(* IEC 61131-3 sources: volt/packages/volt-lsp-iec/test-corpus/lenze-mid/Device/Plc Logic/Application/A70_MachineModuleSources/MM_MachineControl/ATF_ADS, 5 files *)

(* ---- fc_CheckNumberOfErrorsRegister.pou ---- *)
FUNCTION fc_CheckNumberOfErrorsRegister : bool
VAR_INPUT
	iPositie			: ARRAY[0..CTE.ct_ArraySizeCheckRegister] OF cUDT_ShiftRegister_Positie;
	iPositionToCheck : INT;
	iAmountOfErrors : INT;

END_VAR
VAR
	tAmountError : INT;
	tLastPositionToCheck : INT;
	tIndex : INT;

END_VAR
VAR_IN_OUT
	//ioPositie			: ARRAY[0..CTE.ct_ArraySizeCheckRegister] OF cUDT_ShiftRegister_Positie;

END_VAR
VAR_OUTPUT
	oError	: BOOL;
END_VAR
%LANGUAGE ST
//Init
oError := FALSE;
tLastPositionToCheck := 0;
tAmountError := 0;

tLastPositionToCheck := iPositionToCheck + iAmountOfErrors;

FOR tIndex := iPositionToCheck TO tLastPositionToCheck DO

    IF iPositie[tIndex].Infeed.Cigar_Present_Infeed  THEN
        IF iPositie[tIndex].Outfeed.Cigar_Present_Outfeed = 0 THEN
            tAmountError := tAmountError + 1;
        END_IF;
    END_IF;

    IF tAmountError >= iAmountOfErrors THEN
        oError := TRUE;
        EXIT; //Exit for loop
    END_IF;

END_FOR;

END_FUNCTION

(* ---- fc_MeanValue.pou ---- *)
FUNCTION fc_MeanValue
VAR_INPUT
	iLength						: INT;
	iAcquireNewValue			: BOOL;
	iNewValue					: INT;

END_VAR

VAR_OUTPUT
	oMeanValue					: INT;
END_VAR

VAR
	tIndex						: INT;
	tMean						: DINT;
	tCountToIndexNumber			: INT;

END_VAR

VAR_IN_OUT
	ioValues					: ARRAY[0..50] OF INT;
END_VAR
%LANGUAGE ST
oMeanValue := 0;
tMean := 0;
tCountToIndexNumber := iLength - 2; //count from 0 to length -1, but shift is 1 index less -> -2

FOR tIndex:=tCountToIndexNumber TO 0 BY -1 DO
    ioValues[tIndex + 1] := ioValues[tIndex];
    tMean := tMean + ioValues[tIndex];

    IF tIndex= 0 THEN
        ioValues[0] := iNewValue;
        tMean := tMean + ioValues[tIndex];
    END_IF;

END_FOR;
oMeanValue := DINT_TO_INT(tMean / iLength);

END_FUNCTION

(* ---- fc_ShiftRegister.pou ---- *)
FUNCTION fc_ShiftRegister : bool
VAR_INPUT
END_VAR
VAR
	i: INT;
END_VAR
VAR_IN_OUT
	//ioPositie			: ARRAY[0..CTE.ct_ArraySizeCheckRegister] OF cUDT_ShiftRegister_Positie;
	ioPositie			: ARRAY[0..CTE.ct_ArraySizeCheckRegister] OF cUDT_ShiftRegister_Positie;
END_VAR
%LANGUAGE ST
(*
    Shift register
*)
FOR i := CTE.ct_ArraySizeCheckRegister TO 2 BY -1 DO
    ioPositie[i] := ioPositie[i - 1];
END_FOR;

//Eerste register leegmaken
ioPositie[1] := db_CheckRegister.EmptyCheckRegister;

END_FUNCTION

(* ---- Dryer.pou ---- *)
FUNCTION_BLOCK Dryer
VAR_INPUT
	iGenFlags : UDT_GeneralFlags;
iMachineStarted : Bool;
iSwitchDryer : Bool;
iDryerClosed : Bool;
iStartFeedForward : Bool;
iStopFeedForward : Bool;
iPermissionDownstream : Bool;
iSetPowerHeater1 : Int;
iSetPowerHeater2 : Int;
iSetPowerHeater3 : Int;
iPowerOrAnalog : Bool;
iSpeedForEmptying : INT;

END_VAR
VAR_OUTPUT
	ENO: BOOL;
	oFeedForward : BOOL;
oEnableHeaters : Bool;
oPowerHeater1 : Word;
oPowerHeater2 : Word;
oPowerHeater3 : Word;
oFaultDryerOpened : Bool;

END_VAR
VAR
	tEmptyingCycleInterval : DINT;

	stAuxFeedForward: rs;
	tConditionHeaterTimeOut: BOOL;
	tEnableHeaters: BOOL;
	stActPowerHeater1: INT;
	stActPowerHeater2: INT;
	stActPowerHeater3: INT;
	TMR_DryerOpened: TON;
END_VAR

VAR RETAIN PERSISTENT
	stReFeedForward: R_TRIG;
	TMR_IntervalTimerEmptying: TON;
	stFaultDryerOpened: sr;
	stReStopFeedForward: R_TRIG;
	TMR_HeaterTimeOut: TON;
END_VAR
%LANGUAGE LD
%NETWORK "DONE Network 1: Convert speed to cycle time"
// tEmtyingCycle : (1/(MachineSpeed/60))*1000 gives time in [ms]
EXECUTE(EN := RAIL(), 'tEmptyingCycleInterval:=(60*1000)/TO_DINT(iSpeedForEmptying);
');
%NETWORK "DONE Network 2: Feed forward dryer"
ASSIGN(stAuxFeedForward(SET := iStartFeedForward OR TMR_IntervalTimerEmptying(IN := ASSIGN(NOT(stReFeedForward(CLK := stAuxFeedForward.Q1)), Q => tConditionHeaterTimeOut), PT := OPERAND('DINT_TO_TIME(tEmptyingCycleInterval)')) AND iMachineStarted AND INVERT(stFaultDryerOpened.Q1) AND Mach1.GenFlags.DelayAfterSTO AND INVERT(iGenFlags.DriveIsRunning) AND iPermissionDownstream, RESET1 := stReStopFeedForward(CLK := iStopFeedForward)), Q => oFeedForward);
%NETWORK "DONE Network 3: Enable heaters"
VAR w1 : ANY; w2 : ANY; END_VAR
w1 := TRUE;
TMR_HeaterTimeOut(IN := w1 AND INVERT(LST_InputsOutputs.I133_1_PROX_zero_position_transport_ADS), PT := T#7S);
w2 := w1 AND iGenFlags.EnableAuxDrive AND iPermissionDownstream AND INVERT(TMR_HeaterTimeOut.Q) AND iSwitchDryer;
ASSIGN(w2, Q => oEnableHeaters);
ASSIGN(w2, Q => tEnableHeaters);
%NETWORK "DONE Network 4: Output power heater 1"
VAR w3 : ANY; w4 : ANY; END_VAR
w3 := True;
MOVE(EN := w3 AND INVERT(tEnableHeaters), 0, OUT => stActPowerHeater1);
w4 := w3 AND tEnableHeaters;
ADD(EN := w4 AND LST_General.Imp100ms, stActPowerHeater1, 10, OUT => stActPowerHeater1);
MOVE(EN := GT(EN := w4, stActPowerHeater1, iSetPowerHeater1).OUT, iSetPowerHeater1, OUT => stActPowerHeater1);
EXECUTE(EN := w3 AND INVERT(iPowerOrAnalog), 'oPowerHeater1:=INT_TO_WORD(stActPowerHeater1*27648/1000);

');
MOVE(EN := w3 AND iPowerOrAnalog, OPERAND('INT_TO_WORD(stActPowerHeater1)'), OUT => oPowerHeater1);
%NETWORK "DONE Network 5: Output power heater 2"
VAR w5 : ANY; w6 : ANY; END_VAR
w5 := True;
MOVE(EN := w5 AND INVERT(tEnableHeaters), 0, OUT => stActPowerHeater2);
w6 := w5 AND tEnableHeaters;
ADD(EN := w6 AND LST_General.Imp100ms, stActPowerHeater2, 10, OUT => stActPowerHeater2);
MOVE(EN := GT(EN := w6, stActPowerHeater2, iSetPowerHeater2).OUT, iSetPowerHeater2, OUT => stActPowerHeater2);
EXECUTE(EN := w5 AND INVERT(iPowerOrAnalog), 'oPowerHeater2:=INT_TO_WORD(stActPowerHeater2*27648/1000);

');
MOVE(EN := w5 AND iPowerOrAnalog, OPERAND('INT_TO_WORD(stActPowerHeater2)'), OUT => oPowerHeater2);
%NETWORK "DONE Network 6: Output power heater 3"
VAR w7 : ANY; w8 : ANY; END_VAR
w7 := True;
MOVE(EN := w7 AND INVERT(tEnableHeaters), 0, OUT => stActPowerHeater3);
w8 := w7 AND tEnableHeaters;
ADD(EN := w8 AND LST_General.Imp100ms, stActPowerHeater3, 10, OUT => stActPowerHeater3);
MOVE(EN := GT(EN := w8, stActPowerHeater3, iSetPowerHeater3).OUT, iSetPowerHeater3, OUT => stActPowerHeater3);
EXECUTE(EN := w7 AND INVERT(iPowerOrAnalog), 'oPowerHeater3:=INT_TO_WORD(stActPowerHeater3*27648/1000);

');
MOVE(EN := w7 AND iPowerOrAnalog, OPERAND('INT_TO_WORD(stActPowerHeater3)'), OUT => oPowerHeater3);
%NETWORK "DONE Network 37: Fault: dryer opened"
ASSIGN(stFaultDryerOpened(SET1 := TMR_DryerOpened(IN := iMachineStarted AND iSwitchDryer AND INVERT(iDryerClosed) AND INVERT(stFaultDryerOpened.Q1), PT := T#5S), RESET := iGenFlags.StartFlag), Q => oFaultDryerOpened);
%NETWORK
ASSIGN(RAIL(), Q => ENO);

END_FUNCTION_BLOCK

(* ---- TrayFiller.pou ---- *)
FUNCTION_BLOCK TrayFiller
VAR_INPUT
	iGenFlags : UDT_GeneralFlags;
iMachineStarted : Bool;
iButtonChangeTray : Bool;
iButtonTrayDown : Bool;
iButtonTrayUp : Bool;
iCigarAtCrossover : Bool;
iStartFeedForward : Bool;
iStopFeedForward : Bool;
iCigarAtInpusher : Bool;
iRpsInpusher : Bool;
iEpsInpusher : Bool;
iGuardInpusher : Bool;
iPsElevatorUp : Bool;
iPsElevatorDown : Bool;
iPulseCounterElevator : Bool;
iFcGuardTrayOnElev : Bool;
iRowHeight : Int;
iSetNumberOfRows : Int;
iInitialDescentValue : Int;
iLightCurtainInpusher : Bool;
iLightCurtainElevator : Bool;
iPsInfeedConvAtInit : Bool;
iPsInfeedConvAtElev : Bool;
iFcGuardTrayFromElev : Bool;
iFcOutfeedConvFull : Bool;
iTestProd : Bool;

END_VAR
VAR_OUTPUT
	oValveInpusher : BOOL;
oValveTiltInpusher : Bool;
oFeedForwardMotor : Bool;
oElevatorMotorUp : Bool;
oElevatorMotorDown : Bool;
oElevatorMotorBrake : Bool;
oOutfeedMotorFwd : Bool;
oInfeedMotorFwd : Bool;
oInfeedMotorRev : Bool;

END_VAR
VAR
	stRestposition : BOOL;
stInpushingRow : Bool;
stDecendTray : Bool;
stTrayDecended : Bool;
stTiltInpusher : Bool;
stReturnInpusher : Bool;
stLowerInpusher : Bool;
stMoveElevatorUp : Bool;
stMoveElevatorDown : Bool;
stSrCigarAtEndBeforeLast : Bool;
stSrCigarAtEnd : Bool;
stReStopFeedForward : r_trig;
stAuxFeedForward : RS;
stRePulseCounter : r_trig;
stFePulseCounter : F_TRIG;
stFaultInpusherBlocked : SR;
stFaultPositionTray : SR;
stActHeightElevator : Int;
stLightCurtainInterruptedBeforeStart : Bool;
stLightCurtainInterruptedDuringInpushing : Bool;
stElevatorAtBottom : Bool;
stOutfeedTray : Bool;
stOutfeedConvFull : Bool;
stTrayFaultOutfeeding : Bool;
stTrayFedOut : Bool;
stElevatorAtTop : Bool;
stInfeedTray : Bool;
bReturnInfeedConv : Bool;
bFaultOutfeeding : Bool;
bRecoverFromLightCurtainInterrupted : Bool;
TMR_InpusherDown : ton;
TMR_DelayReturnInfeed : ton;
TMR_DelayDescend : ton;
TMR_InpusherTilted : ton;
TMR_DelayEmptying : ton;
TMR_DelayFaultOutfeed : ton;
TMR_DelayTrayFedOut : ton;
TOdoTEst : ctd;

	tBool: BOOL;
	tInt: INT;
	SET_stFaultPositionTray:BOOL;
END_VAR

VAR_IN_OUT
	ioActNumberOfRows: INT;
END_VAR
%LANGUAGE LD
%NETWORK "DONE NETWORK 1: Condition: Reset all"
ASSIGN(LST_General.FirstCycle, Q_SET => stRestposition, Q_RESET => bReturnInfeedConv, Q_RESET => stInpushingRow, Q_RESET => stDecendTray, Q_RESET => stTrayDecended, Q_RESET => stTiltInpusher, Q_RESET => stReturnInpusher, Q_RESET => stLowerInpusher, Q_RESET => stMoveElevatorUp, Q_RESET => stMoveElevatorDown, Q_RESET => stElevatorAtBottom, Q_RESET => stOutfeedTray, Q_RESET => stTrayFedOut, Q_RESET => stElevatorAtTop, Q_RESET => stInfeedTray, Q_RESET => stLightCurtainInterruptedBeforeStart, Q_RESET => stLightCurtainInterruptedDuringInpushing, Q_RESET => stTrayFaultOutfeeding, Q_RESET => bRecoverFromLightCurtainInterrupted, Q_RESET => stSrCigarAtEnd);
%NETWORK "DONE NETWORK 2: Condition: Rest position"
VAR w1 : ANY; END_VAR
w1 := TMR_InpusherDown(IN := stLowerInpusher, PT := T#500MS) OR stInfeedTray AND iPsInfeedConvAtElev OR stLightCurtainInterruptedBeforeStart AND iLightCurtainInpusher AND iGenFlags.StartFlag;
ASSIGN(w1, Q_SET => stRestposition, Q_RESET => stLowerInpusher, Q_RESET => stInfeedTray, Q_RESET => stLightCurtainInterruptedBeforeStart);
ASSIGN(w1 AND INVERT(iFcGuardTrayOnElev) AND iTestProd, Q_SET => Trayfiller_Data.Alarms.AlmTrayInfeeding);
%NETWORK "TODO NETWORK 3: Condition: Set infeed conveyor at init position"
VAR w2 : ANY; END_VAR
w2 := True;
ASSIGN(w2 AND bReturnInfeedConv AND iPsInfeedConvAtInit, Q_RESET => bReturnInfeedConv);
ASSIGN(w2 AND iGenFlags.StartFlag AND (iFcGuardTrayOnElev OR INVERT(iTestProd)), Q_RESET => Trayfiller_Data.Alarms.AlmTrayInfeeding);
%NETWORK "DONE NETWORK 4: Delay return infeed conveyor"
TMR_DelayReturnInfeed(IN := bReturnInfeedConv, PT := T#500MS);
%NETWORK "DONE NETWORK 5: Condition: Inpushing row"
ASSIGN(stRestposition AND stSrCigarAtEnd AND INVERT(stFaultPositionTray.Q1), Q_SET => stInpushingRow, Q_RESET => stRestposition);
%NETWORK "TODO NETWORK 6: Condition: Light curtain inpusher interrupted before start"
ASSIGN((stInpushingRow OR stRestposition AND stSrCigarAtEndBeforeLast) AND INVERT(iLightCurtainInpusher) AND iRpsInpusher, Q_SET => stLightCurtainInterruptedBeforeStart, Q_RESET => stInpushingRow);
%NETWORK "TODO NETWORK 7: Condition: Decend tray"
ASSIGN(ADD(EN := (TMR_DelayDescend(IN := stInpushingRow AND iLightCurtainInpusher AND iEpsInpusher, PT := T#500MS) OR stLightCurtainInterruptedDuringInpushing AND iLightCurtainInpusher AND iGenFlags.StartFlag) AND INVERT(stFaultInpusherBlocked.Q1), ioActNumberOfRows, 1, OUT => ioActNumberOfRows), Q_SET => stDecendTray, Q_RESET => stInpushingRow, Q_RESET => stLightCurtainInterruptedDuringInpushing, Q_RESET => stSrCigarAtEndBeforeLast, Q_RESET => stSrCigarAtEnd);
%NETWORK "TODO NETWORK 8: Condition: Light curtain inpusher interrupted during inpushing"
ASSIGN(stInpushingRow AND INVERT(iLightCurtainInpusher) AND INVERT(iRpsInpusher), Q_SET => stLightCurtainInterruptedDuringInpushing, Q_RESET => stInpushingRow, Q_RESET => bRecoverFromLightCurtainInterrupted);
%NETWORK "TODO NETWORK 9: Condition: Tray decend"
VAR w3 : ANY; w4 : ANY; w5 : ANY; END_VAR
w3 := True;
w4 := w3 AND True;
w5 := w4 AND iPulseCounterElevator;
ASSIGN(stRePulseCounter(CLK := w5), Q => tBool);
ASSIGN(stFePulseCounter(CLK := w5), Q_SET => tBool);
ADD(EN := w4 AND tBool AND (stDecendTray OR stTrayDecended OR stTiltInpusher), stActHeightElevator, 5, OUT => stActHeightElevator);
ASSIGN(BRANCH_SHORTCIRCUIT(FEED := ADD(EN := MUL(EN := w3 AND stDecendTray, ioActNumberOfRows, iRowHeight, OUT => tInt), tInt, iInitialDescentValue, OUT => tInt), GE(EN := RAIL(), stActHeightElevator, tInt).OUT, iPsElevatorDown), Q_SET => stTrayDecended, Q_RESET => stDecendTray);
%NETWORK "TODO NETWORK 10: Condition: Tilt inpusher"
ASSIGN(stTrayDecended, Q_SET => stTiltInpusher, Q_RESET => stTrayDecended, Q_SET => bReturnInfeedConv);
%NETWORK "TODO NETWORK 11: Condition: Return inpusher"
ASSIGN(TMR_InpusherTilted(IN := stTiltInpusher, PT := T#500MS), Q_SET => stReturnInpusher, Q_RESET => stTiltInpusher);
%NETWORK "TODO NETWORK 12: Condition: Lower inpusher"
ASSIGN(LT(EN := stReturnInpusher AND iRpsInpusher, ioActNumberOfRows, iSetNumberOfRows).OUT AND INVERT(iPsElevatorDown) AND INVERT(stFaultInpusherBlocked.Q1), Q_SET => stLowerInpusher, Q_RESET => stReturnInpusher, Q_RESET => bRecoverFromLightCurtainInterrupted);
%NETWORK "TODO NETWORK 13: Condition: Move elevator down"
ASSIGN(BRANCH_SHORTCIRCUIT(BRANCH_SHORTCIRCUIT(FEED := stReturnInpusher AND iRpsInpusher, GE(EN := RAIL(), ioActNumberOfRows, iSetNumberOfRows).OUT, iPsElevatorDown) AND INVERT(stFaultInpusherBlocked.Q1) AND iMachineStarted, stOutfeedConvFull AND iGenFlags.StartFlag, TMR_DelayEmptying(IN := stRestposition AND iGenFlags.DelayAfterEmergStop AND iPsElevatorDown, PT := T#2S)), Q_SET => stMoveElevatorDown, Q_RESET => stReturnInpusher, Q_RESET => stOutfeedConvFull, Q_RESET => stRestposition);
%NETWORK "TODO NETWORK 14: Condition: Elevator at bottom"
ASSIGN(stMoveElevatorDown AND iPsElevatorDown OR stTrayFaultOutfeeding AND iGenFlags.StartFlag OR stElevatorAtTop AND oElevatorMotorDown AND iPsElevatorDown AND iButtonTrayDown, Q_SET => stElevatorAtBottom, Q_RESET => stMoveElevatorDown, Q_RESET => stTrayFaultOutfeeding, Q_RESET => stElevatorAtTop, Q_SET => bReturnInfeedConv);
%NETWORK "TODO NETWORK 15: Condition: Outfeed conveyor full"
ASSIGN(stElevatorAtBottom AND iMachineStarted AND iFcOutfeedConvFull, Q_SET => stOutfeedConvFull, Q_RESET => stElevatorAtBottom);
%NETWORK "TODO NETWORK 16: Condition: Outfeed tray"
ASSIGN(stElevatorAtBottom AND iMachineStarted AND INVERT(iFcOutfeedConvFull), Q_SET => stOutfeedTray, Q_RESET => stElevatorAtBottom, Q_SET => bReturnInfeedConv);
%NETWORK "TODO NETWORK 17: Condition: Fault Outfeeding"
ASSIGN(TMR_DelayFaultOutfeed(IN := stOutfeedTray AND (INVERT(iFcGuardTrayFromElev) AND INVERT(iFcOutfeedConvFull) OR iFcGuardTrayFromElev AND iFcOutfeedConvFull) AND iTestProd, PT := T#7S), Q_SET => stTrayFaultOutfeeding, Q_RESET => stOutfeedTray, Q_RESET => bFaultOutfeeding);
%NETWORK "TODO NETWORK 18: Condition: Tray fed out"
ASSIGN(TMR_DelayTrayFedOut(IN := stOutfeedTray AND INVERT(iFcGuardTrayFromElev) AND (iFcOutfeedConvFull OR INVERT(iTestProd)), PT := T#500MS), Q_SET => stTrayFedOut, Q_RESET => stOutfeedTray, Q_RESET => bFaultOutfeeding);
%NETWORK "TODO NETWORK 19: Condition: Move elevator up"
ASSIGN(stTrayFedOut AND iMachineStarted, Q_SET => stMoveElevatorUp, Q_RESET => stTrayFedOut);
%NETWORK "TODO NETWORK 20: Condition: Elevator at top"
ASSIGN(MOVE(EN := MOVE(EN := stMoveElevatorUp AND iPsElevatorUp, 0, OUT => ioActNumberOfRows), 0, OUT => stActHeightElevator), Q_SET => stElevatorAtTop, Q_RESET => stMoveElevatorUp);
%NETWORK "TODO NETWORK 21: Condition: Infeed tray"
ASSIGN(stElevatorAtTop AND (INVERT(iFcGuardTrayOnElev) OR INVERT(iTestProd)) AND INVERT(bReturnInfeedConv), Q_SET => stInfeedTray, Q_RESET => stElevatorAtTop);
%NETWORK "TODO NETWORK 22: Condition: Light curtain elevator interrupted "
VAR w6 : ANY; END_VAR
w6 := True;
ASSIGN(w6 AND True AND (oElevatorMotorUp OR oElevatorMotorDown) AND INVERT(iLightCurtainElevator), Q_SET => Trayfiller_Data.Alarms.AlmLightCurtainElevator);
ASSIGN(w6 AND iGenFlags.StartFlag AND iLightCurtainElevator, Q_RESET => Trayfiller_Data.Alarms.AlmLightCurtainElevator);
%NETWORK "TODO NETWORK 23: Output: Fault inpusher blocked"
ASSIGN(stFaultInpusherBlocked(SET1 := iGenFlags.DelayAfterEmergStop AND INVERT(iGuardInpusher), RESET := iGenFlags.StartFlag), Q => Trayfiller_Data.Alarms.AlmInpusherBlocked);
%NETWORK "TODO NETWORK 24: Output: Fault position tray"
ASSIGN(stFaultPositionTray(SET1 := iGenFlags.DelayAfterEmergStop AND (stSrCigarAtEndBeforeLast OR stSrCigarAtEnd) AND INVERT(iFcGuardTrayOnElev) AND iTestProd, RESET := iGenFlags.StartFlag OR stMoveElevatorUp), Q => Trayfiller_Data.Alarms.AlmTrayPosition);
%NETWORK "TODO NETWORK 25: Output: Fault outfeed conveyor full"
ASSIGN(iGenFlags.DelayAfterEmergStop AND stOutfeedConvFull, Q => Trayfiller_Data.Alarms.AlmOutfeedFull);
%NETWORK "TODO NETWORK 26: Output: Fault Tray outfeeding"
ASSIGN(iGenFlags.DelayAfterEmergStop AND stTrayFaultOutfeeding, Q => Trayfiller_Data.Alarms.AlmOutfeeding);
%NETWORK "TODO NETWORK 27: Output: Permission upstream"
ASSIGN(((INVERT(stSrCigarAtEndBeforeLast) OR stRestposition) AND INVERT(stSrCigarAtEnd) OR stInpushingRow) AND INVERT(stFaultInpusherBlocked.Q1) AND INVERT(stFaultPositionTray.Q1) AND INVERT(stLightCurtainInterruptedBeforeStart) AND INVERT(stLightCurtainInterruptedDuringInpushing), Q => Trayfiller_Data.commInterface.Permission);
%NETWORK "TODO NETWORK 28: Output: lightcurtain inpusher interrupted"
ASSIGN(stLightCurtainInterruptedBeforeStart OR stLightCurtainInterruptedDuringInpushing, Q => Trayfiller_Data.Alarms.AlmLightCurtainInpusher);
%NETWORK "TODO NETWORK 29: Output: Valve inpusher"
ASSIGN(iGenFlags.EnablePneumEStop AND (stInpushingRow OR (stDecendTray OR stTrayDecended OR stTiltInpusher) AND INVERT(bRecoverFromLightCurtainInterrupted)), Q => oValveInpusher);
%NETWORK "TODO NETWORK 30: Output: Valve tilt inpusher"
ASSIGN(iGenFlags.EnablePneumEStop AND (stTiltInpusher OR stReturnInpusher OR stLightCurtainInterruptedDuringInpushing OR stDecendTray AND bRecoverFromLightCurtainInterrupted), Q => oValveTiltInpusher);
%NETWORK "TODO NETWORK 31: Output: Feed forward motor"
ASSIGN(stAuxFeedForward(SET := iStartFeedForward AND (iCigarAtCrossover OR INVERT(iTestProd)), RESET1 := ASSIGN(stReStopFeedForward(CLK := iStopFeedForward), Q => tBool)) AND iGenFlags.DelayAfterEmergStop, Q => oFeedForwardMotor);
%NETWORK "TODO NETWORK 32: TODo test count down"
ASSIGN(TOdoTEst(CD := tBool, LOAD := stSrCigarAtEnd, PV := 30), Q => ToDo.CounterCigarAtEnd);
%NETWORK "TODO NETWORK 33: Aux marker: Cigar detection register"
VAR w7 : ANY; w8 : ANY; END_VAR
w7 := tBool;
w8 := w7 AND stSrCigarAtEndBeforeLast;
ASSIGN(w8, Q_SET => stSrCigarAtEnd);
ASSIGN(w8 AND LST_General.AlwaysOff, Q_RESET => stSrCigarAtEndBeforeLast);
ASSIGN(w7 AND (iCigarAtInpusher OR INVERT(iTestProd) AND ToDo.CounterCigarAtEnd) AND iRpsInpusher AND INVERT(stLowerInpusher), Q_SET => stSrCigarAtEndBeforeLast);
%NETWORK "TODO NETWORK 34: Ouput: Stop feedforward while inpushing"
VAR w9 : ANY; END_VAR
w9 := iGenFlags.DelayAfterEmergStop;
ASSIGN(w9 AND (stMoveElevatorUp OR INVERT(stDecendTray) AND iButtonTrayUp) AND INVERT(iPsElevatorUp) AND INVERT(oElevatorMotorDown) AND INVERT(Trayfiller_Data.Alarms.AlmLightCurtainElevator), Q => oElevatorMotorUp);
ASSIGN(w9 AND (stMoveElevatorDown OR stDecendTray OR iButtonTrayDown) AND INVERT(iPsElevatorDown) AND INVERT(oElevatorMotorUp) AND INVERT(Trayfiller_Data.Alarms.AlmLightCurtainElevator), Q => oElevatorMotorDown);
ASSIGN(w9 AND (oElevatorMotorUp OR oElevatorMotorDown), Q => oElevatorMotorBrake);
%NETWORK "TODO NETWORK 35: Ouput: Stop feedforward while inpushing"
ASSIGN(stInpushingRow AND INVERT(iEpsInpusher), Q => Trayfiller_Data.commInterface.HoldFeedFwd);
%NETWORK "TODO NETWORK 36: Output: Infeed conveyor"
VAR w10 : ANY; END_VAR
w10 := iGenFlags.DelayAfterEmergStop AND (Mach1.GenFlags.RunAuto OR Mach1.GenFlags.RunMan);
ASSIGN(w10 AND stInfeedTray AND INVERT(iPsInfeedConvAtElev) AND INVERT(oInfeedMotorRev), Q => oInfeedMotorFwd);
ASSIGN(w10 AND TMR_DelayReturnInfeed.Q AND INVERT(Trayfiller_Data.Alarms.AlmTrayInfeeding) AND INVERT(iPsInfeedConvAtInit) AND INVERT(oInfeedMotorFwd), Q => oInfeedMotorRev);
%NETWORK "TODO NETWORK 37: Output: Outfeed conveyor"
ASSIGN(iGenFlags.DelayAfterEmergStop AND stOutfeedTray AND Mach1.GenFlags.EnableAuxDrive, Q => oOutfeedMotorFwd);

END_FUNCTION_BLOCK
